END_FUNCTION_BLOCK

// K2/std12k5/TestIm/TestImAlg
	{attribute 'symbol' := 'none'}
FUNCTION_BLOCK TestImAlg EXTENDS BaseAlgoritm
VAR_INPUT
END_VAR
VAR_OUTPUT
END_VAR
VAR
END_VAR

SUPER^();
BlockIm(im:=im.TEN_MB,block:=((BlockOpcControl(block:=FALSE)) OR (im.CMN.onStatus = statusDualInput.STATUS_ERROR) OR (im.CMN.onStatus = statusDualInput.STATUS_NOTDEFINED) OR 
(im.CMN.onStatus = statusDualInput.STATUS_OFF) OR (im.CMN.onStatus = statusDualInput.STATUS_TRANSITIONAL) ));
IF	(im.CMN.onStatus = statusDualInput.STATUS_OFF) AND (im.TEN_MB.onStatus = statusDualInput.STATUS_on) THEN
	im.TEN_MB.off();
END_IF
BlockIm(im:=im.nu.nu1,block:=((BlockOpcControl(block:=FALSE)) OR (im.PNS.onStatus = statusDualInput.STATUS_ERROR) OR (im.pns.onStatus = statusDualInput.STATUS_NOTDEFINED) OR 
(im.pns.onStatus = statusDualInput.STATUS_OFF) OR (im.pns.onStatus = statusDualInput.STATUS_TRANSITIONAL) ));
BlockIm(im:=im.nu.nu2,block:=((BlockOpcControl(block:=FALSE)) OR (im.PNS.onStatus = statusDualInput.STATUS_ERROR) OR (im.pns.onStatus = statusDualInput.STATUS_NOTDEFINED) OR 
(im.pns.onStatus = statusDualInput.STATUS_OFF) OR (im.pns.onStatus = statusDualInput.STATUS_TRANSITIONAL) ));
IF	(im.pns.onStatus = statusDualInput.STATUS_OFF) AND ((im.nu.nu1.onStatus = statusDualInput.STATUS_on) OR (im.nu.nu2.onStatus = statusDualInput.STATUS_on)) THEN
	im.nu.off();
END_IF

METHOD PUBLIC reset
VAR_INPUT
END_VAR
SUPER^.reset();
BlockOpcControl(block:=TRUE);
IF	(algmanager.mode <> modegpa.MODE_AO) AND (algmanager.mode <> modegpa.MODE_NO) AND (algmanager.mode <> modegpa.MODE_EO) THEN
	algManager.setMode(nMode:=ModeGpa.MODE_STOP);
END_IF
im.PNS.DisableOpcControl();
im.nu.nu1.DisableOpcControl();
im.nu.nu2.DisableOpcControl();
im.CMN.DisableOpcControl();
im.TEN_MB.DisableOpcControl();
IF	im.PNS.onStatus = statusDualInput.STATUS_ON THEN
	im.PNS.off();
END_IF
IF	im.nu.nu1.onStatus = statusDualInput.STATUS_ON THEN
	im.nu.nu1.off();
END_IF
IF	im.nu.nu2.onStatus = statusDualInput.STATUS_ON THEN
	im.nu.nu2.off();
END_IF
IF	im.cmn.onStatus = statusDualInput.STATUS_ON THEN
	im.cmn.off();
END_IF
IF	im.TEN_MB.onStatus = statusDualInput.STATUS_ON THEN
	im.TEN_MB.off();
END_IF
END_METHOD

METHOD PUBLIC run
VAR_INPUT
END_VAR
SUPER^.run();
BlockOpcControl(block:=FALSE);
algManager.setMode(nMode:=ModeGpa.MODE_TESTIM);

im.mv.DisableOpcControl ();
im.kran1.DisableOpcControl ();
im.kran2.DisableOpcControl ();
im.kran3.DisableOpcControl ();
im.kran3b.DisableOpcControl ();
im.kran4.DisableOpcControl ();
im.kran5.DisableOpcControl ();
END_METHOD

END_FUNCTION_BLOCK

// K1/std12k5/Start_ALG/Start_NO
{attribute 'symbol' := 'none'}
FUNCTION_BLOCK Start_NO EXTENDS StepBySteapAlgoritm
VAR_INPUT
END_VAR
	
VAR_OUTPUT
	{attribute 'symbol' := 'read'}
	Start_Prov_Pusk:		Question(table:=ADR(ObjectTable)):=			(AnswerVariants:=(Answers.ANS_YES OR Answers.ANS_NO));
END_VAR
VAR
	Alg_Start_reset:	ph_algoritm (table:=ADR(phasesTable)):=		(phaseNumber:=0, Im:=algoritms.no, act:=PhaseAlgoritmAction.run, waitCompletion:=FALSE);
END_VAR

SUPER^();
IF	NOT Alg_Start_reset.start THEN
	Start_Prov_Pusk.ask ();
END_IF
IF	(Start_Prov_Pusk.answer=Answers.ANS_YES) THEN
	algoritms.no.CanRun:=TRUE;
	Alg_Start_reset.run ();
	Start_Prov_Pusk.reset ();
	reset ();
ELSIF	(Start_Prov_Pusk.answer=Answers.ANS_NO) THEN
		algoritms.no.CanRun:=FALSE;
		Start_Prov_Pusk.reset ();
		reset ();
END_IF

METHOD PUBLIC reset
VAR_INPUT
END_VAR
SUPER^.reset();
Start_Prov_Pusk.reset ();
END_METHOD

END_FUNCTION_BLOCK

// K2/std12k5/Start_ALG/Start_NO
{attribute 'symbol' := 'none'}
FUNCTION_BLOCK Start_NO EXTENDS StepBySteapAlgoritm
VAR_INPUT
END_VAR
	
VAR_OUTPUT
	{attribute 'symbol' := 'read'}
	Start_Prov_Pusk:		Question(table:=ADR(ObjectTable)):=			(AnswerVariants:=(Answers.ANS_YES OR Answers.ANS_NO));
END_VAR
VAR
	Alg_Start_reset:	ph_algoritm (table:=ADR(phasesTable)):=		(phaseNumber:=0, Im:=algoritms.no, act:=PhaseAlgoritmAction.run, waitCompletion:=FALSE);
END_VAR

SUPER^();
IF	NOT Alg_Start_reset.start THEN
	Start_Prov_Pusk.ask ();
END_IF
IF	(Start_Prov_Pusk.answer=Answers.ANS_YES) THEN
	algoritms.no.CanRun:=TRUE;
	Alg_Start_reset.run ();
	Start_Prov_Pusk.reset ();
	reset ();
ELSIF	(Start_Prov_Pusk.answer=Answers.ANS_NO) THEN
		algoritms.no.CanRun:=FALSE;
		Start_Prov_Pusk.reset ();
		reset ();
END_IF

METHOD PUBLIC reset
VAR_INPUT
END_VAR
SUPER^.reset();
Start_Prov_Pusk.reset ();
END_METHOD

END_FUNCTION_BLOCK

// K1/std12k5/Start_ALG/Start_AO
{attribute 'symbol' := 'none'}
FUNCTION_BLOCK Start_AO EXTENDS StepBySteapAlgoritm
VAR_INPUT
END_VAR
	
VAR_OUTPUT
	{attribute 'symbol' := 'read'}
	Start_Prov_Pusk:		Question(table:=ADR(ObjectTable)):=			(AnswerVariants:=(Answers.ANS_YES OR Answers.ANS_NO));
END_VAR
VAR
	Alg_Start_reset:	ph_algoritm (table:=ADR(phasesTable)):=		(phaseNumber:=0, Im:=algoritms.ao, act:=PhaseAlgoritmAction.run, waitCompletion:=FALSE);
END_VAR

SUPER^();
IF	NOT Alg_Start_reset.start THEN
	Start_Prov_Pusk.ask ();
END_IF
IF	(Start_Prov_Pusk.answer=Answers.ANS_YES) THEN
	algoritms.ao.CanRun:=TRUE;
	Alg_Start_reset.run ();
	Start_Prov_Pusk.reset ();
	reset ();
ELSIF	(Start_Prov_Pusk.answer=Answers.ANS_NO) THEN
		algoritms.ao.CanRun:=FALSE;
		Start_Prov_Pusk.reset ();
		reset ();
END_IF

METHOD PUBLIC reset
VAR_INPUT
END_VAR
SUPER^.reset();
Start_Prov_Pusk.reset ();
END_METHOD

END_FUNCTION_BLOCK

// K2/std12k5/Start_ALG/Start_AO
{attribute 'symbol' := 'none'}
FUNCTION_BLOCK Start_AO EXTENDS StepBySteapAlgoritm
VAR_INPUT
END_VAR
	
VAR_OUTPUT
	{attribute 'symbol' := 'read'}
	Start_Prov_Pusk:		Question(table:=ADR(ObjectTable)):=			(AnswerVariants:=(Answers.ANS_YES OR Answers.ANS_NO));
END_VAR
VAR
	Alg_Start_reset:	ph_algoritm (table:=ADR(phasesTable)):=		(phaseNumber:=0, Im:=algoritms.ao, act:=PhaseAlgoritmAction.run, waitCompletion:=FALSE);
END_VAR

SUPER^();
IF	NOT Alg_Start_reset.start THEN
	Start_Prov_Pusk.ask ();
END_IF
IF	(Start_Prov_Pusk.answer=Answers.ANS_YES) THEN
	algoritms.ao.CanRun:=TRUE;
	Alg_Start_reset.run ();
	Start_Prov_Pusk.reset ();
	reset ();
ELSIF	(Start_Prov_Pusk.answer=Answers.ANS_NO) THEN
		algoritms.ao.CanRun:=FALSE;
		Start_Prov_Pusk.reset ();
		reset ();
END_IF

METHOD PUBLIC reset
VAR_INPUT
END_VAR
SUPER^.reset();
Start_Prov_Pusk.reset ();
END_METHOD

END_FUNCTION_BLOCK

// K1/std12k5/Logic/SIP_PS
{attribute 'symbol' := 'none'}
FUNCTION_BLOCK SIP_PS EXTENDS BaseIM
VAR_INPUT
	Ai:REFERENCE TO AISource;
END_VAR
VAR_OUTPUT
END_VAR
VAR
	
END_VAR

SUPER^();
IF __ISVALIDREF(Ai) THEN
	
	IF 	ai.interval=statusAi.NOTRELIABLE THEN
		statusSet.setBit (bitNum:=0,value:=1);
	ELSE
		statusSet.setBit (bitNum:=0,value:=0);
	END_IF
END_IF

END_FUNCTION_BLOCK

// K2/std12k5/Logic/SIP_PS
{attribute 'symbol' := 'none'}
FUNCTION_BLOCK SIP_PS EXTENDS BaseIM
VAR_INPUT
	Ai:REFERENCE TO AISource;
END_VAR
VAR_OUTPUT
END_VAR
VAR
	
END_VAR

SUPER^();
IF __ISVALIDREF(Ai) THEN
	
	IF 	ai.interval=statusAi.NOTRELIABLE THEN
		statusSet.setBit (bitNum:=0,value:=1);
	ELSE
		statusSet.setBit (bitNum:=0,value:=0);
	END_IF
END_IF

END_FUNCTION_BLOCK

// K1/std12k5/Ystavki/SIp_Yst
	{attribute 'symbol' := 'none'}
FUNCTION_BLOCK SIp_Yst EXTENDS Baseobject
VAR_INPUT
	{attribute 'symbol' := 'readwright'}
	Yst_izm:ARRAY [0..17] OF UINT;
END_VAR
VAR_OUTPUT
	{attribute 'symbol' := 'read'}
	Yst:ARRAY [0..17] OF UINT;
	
END_VAR
VAR
	flag:BOOL;
	flag2:bool;
	i:uINT;
END_VAR

SUPER^();

FOR i:=0 TO 17 DO
	IF 	(Yst_izm [i] <> Yst [i]) AND (Yst_izm [i] >=0) AND (Yst_izm [i] <=17) THEN
		Yst[i] := Yst_izm [i];
		SaveToFile();
	END_IF	
	
	IF	(Yst_izm [i] = 0) AND (Yst [i] = 0) AND NOT flag AND flag2 THEN
		Yst [i] := 10;
		Yst_izm [i] := Yst [i];
		SaveToFile();
	END_IF


	
END_FOR
IF flag2 THEN
	flag:=TRUE;
END_IF
flag2:=TRUE;

METHOD PROTECTED readPersistent
VAR_INPUT
END_VAR
Yst_izm [0]:=STRING_TO_UINT(readValue());
Yst_izm [1]:=STRING_TO_UINT(readValue());
Yst_izm [2]:=STRING_TO_UINT(readValue());
Yst_izm [3]:=STRING_TO_UINT(readValue());
Yst_izm [4]:=STRING_TO_UINT(readValue());
Yst_izm [5]:=STRING_TO_UINT(readValue());
Yst_izm [6]:=STRING_TO_UINT(readValue());
Yst_izm [7]:=STRING_TO_UINT(readValue());
Yst_izm [8]:=STRING_TO_UINT(readValue());
Yst_izm [9]:=STRING_TO_UINT(readValue());
Yst_izm [10]:=STRING_TO_UINT(readValue());
Yst_izm [11]:=STRING_TO_UINT(readValue());
Yst_izm [12]:=STRING_TO_UINT(readValue());
Yst_izm [13]:=STRING_TO_UINT(readValue());
Yst_izm [14]:=STRING_TO_UINT(readValue());
Yst_izm [15]:=STRING_TO_UINT(readValue());
Yst_izm [16]:=STRING_TO_UINT(readValue());
Yst_izm [17]:=STRING_TO_UINT(readValue());
END_METHOD

METHOD PROTECTED writePersistent
VAR_INPUT
END_VAR

writeValue(value:= UINT_TO_STRING(Yst [0]),'Наработка');
writeValue(value:= UINT_TO_STRING(Yst [1]),'Наработка');
writeValue(value:= UINT_TO_STRING(Yst[2]),'Наработка');
writeValue(value:= UINT_TO_STRING(Yst [3]),'Наработка');

writeValue(value:= UINT_TO_STRING(Yst [4]),'Наработка');
writeValue(value:= UINT_TO_STRING(Yst [5]),'Наработка');
writeValue(value:= UINT_TO_STRING(Yst[6]),'Наработка');
writeValue(value:= UINT_TO_STRING(Yst [7]),'Наработка');

writeValue(value:= UINT_TO_STRING(Yst[8]),'Наработка');
writeValue(value:= UINT_TO_STRING(Yst [9]),'Наработка');
writeValue(value:= UINT_TO_STRING(Yst [10]),'Наработка');
writeValue(value:= UINT_TO_STRING(Yst [11]),'Наработка');

writeValue(value:= UINT_TO_STRING(Yst[12]),'Наработка');
writeValue(value:= UINT_TO_STRING(Yst[13]),'Наработка');
writeValue(value:= UINT_TO_STRING(Yst [14]),'Наработка');
writeValue(value:= UINT_TO_STRING(Yst [15]),'Наработка');
writeValue(value:= UINT_TO_STRING(Yst[16]),'Наработка');
writeValue(value:= UINT_TO_STRING(Yst [17]),'Наработка');
END_METHOD

END_FUNCTION_BLOCK

// K2/std12k5/Ystavki/SIp_Yst
	{attribute 'symbol' := 'none'}
FUNCTION_BLOCK SIp_Yst EXTENDS Baseobject
VAR_INPUT
	{attribute 'symbol' := 'readwright'}
	Yst_izm:ARRAY [0..17] OF UINT;
END_VAR
VAR_OUTPUT
	{attribute 'symbol' := 'read'}
	Yst:ARRAY [0..17] OF UINT;
	
END_VAR
VAR
	flag:BOOL;
	flag2:bool;
	i:uINT;
END_VAR

SUPER^();

FOR i:=0 TO 17 DO
	IF 	(Yst_izm [i] <> Yst [i]) AND (Yst_izm [i] >=0) AND (Yst_izm [i] <=17) THEN
		Yst[i] := Yst_izm [i];
		SaveToFile();
	END_IF	
	
	IF	(Yst_izm [i] = 0) AND (Yst [i] = 0) AND NOT flag AND flag2 THEN
		Yst [i] := 10;
		Yst_izm [i] := Yst [i];
		SaveToFile();
	END_IF


	
END_FOR
IF flag2 THEN
	flag:=TRUE;
END_IF
flag2:=TRUE;

METHOD PROTECTED readPersistent
VAR_INPUT
END_VAR
Yst_izm [0]:=STRING_TO_UINT(readValue());
Yst_izm [1]:=STRING_TO_UINT(readValue());
Yst_izm [2]:=STRING_TO_UINT(readValue());
Yst_izm [3]:=STRING_TO_UINT(readValue());
Yst_izm [4]:=STRING_TO_UINT(readValue());
Yst_izm [5]:=STRING_TO_UINT(readValue());
Yst_izm [6]:=STRING_TO_UINT(readValue());
Yst_izm [7]:=STRING_TO_UINT(readValue());
Yst_izm [8]:=STRING_TO_UINT(readValue());
Yst_izm [9]:=STRING_TO_UINT(readValue());
Yst_izm [10]:=STRING_TO_UINT(readValue());
Yst_izm [11]:=STRING_TO_UINT(readValue());
Yst_izm [12]:=STRING_TO_UINT(readValue());
Yst_izm [13]:=STRING_TO_UINT(readValue());
Yst_izm [14]:=STRING_TO_UINT(readValue());
Yst_izm [15]:=STRING_TO_UINT(readValue());
Yst_izm [16]:=STRING_TO_UINT(readValue());
Yst_izm [17]:=STRING_TO_UINT(readValue());
END_METHOD

METHOD PROTECTED writePersistent
VAR_INPUT
END_VAR

writeValue(value:= UINT_TO_STRING(Yst [0]),'Наработка');
writeValue(value:= UINT_TO_STRING(Yst [1]),'Наработка');
writeValue(value:= UINT_TO_STRING(Yst[2]),'Наработка');
writeValue(value:= UINT_TO_STRING(Yst [3]),'Наработка');

writeValue(value:= UINT_TO_STRING(Yst [4]),'Наработка');
writeValue(value:= UINT_TO_STRING(Yst [5]),'Наработка');
writeValue(value:= UINT_TO_STRING(Yst[6]),'Наработка');
writeValue(value:= UINT_TO_STRING(Yst [7]),'Наработка');

writeValue(value:= UINT_TO_STRING(Yst[8]),'Наработка');
writeValue(value:= UINT_TO_STRING(Yst [9]),'Наработка');
writeValue(value:= UINT_TO_STRING(Yst [10]),'Наработка');
writeValue(value:= UINT_TO_STRING(Yst [11]),'Наработка');

writeValue(value:= UINT_TO_STRING(Yst[12]),'Наработка');
writeValue(value:= UINT_TO_STRING(Yst[13]),'Наработка');
writeValue(value:= UINT_TO_STRING(Yst [14]),'Наработка');
writeValue(value:= UINT_TO_STRING(Yst [15]),'Наработка');
writeValue(value:= UINT_TO_STRING(Yst[16]),'Наработка');
writeValue(value:= UINT_TO_STRING(Yst [17]),'Наработка');
END_METHOD

END_FUNCTION_BLOCK

// K1/std12k5/Narabotka/CMN_
	{attribute 'symbol' := 'none'}
FUNCTION_BLOCK CMN_ EXTENDS nasos
VAR_INPUT
END_VAR
VAR_OUTPUT
		{attribute 'symbol' := 'read'}
	narabotka:UDINT;
		narabotka_:ExtNarabotka (table:=ADR (objectTable)):=(saveInterval:=T#1H);
END_VAR
VAR
	(*timer:RTC;	
	saveTimer:TON:=(PT:=T#600S);
	Narabotka_hour:R_TRIG;
	AvomStartted:R_TRIG;
	narabotka_Izm:UDINT;*)
END_VAR

SUPER^();
narabotka_.started:=onstatus=statusDualInput.STATUS_ON;
narabotka:=(narabotka_.narabotka/3600);
(*
AvomStartted(CLK:=im.CMN.onStatus=statusDualInput.status_on);

	timer.PDT:=UDINT_TO_DT(narabotka_izm);

IF im.CMN.onStatus=statusDualInput.status_on THEN
	narabotka_izm:=DT_TO_UDINT( timer.CDT);
	timer.EN:=TRUE;
ELSE
	timer.EN:=FALSE;
END_IF
narabotka_hour (clk:=(narabotka_izm >=3600));
IF	narabotka_hour.Q THEN
	narabotka:=narabotka+1;
	timer.EN:=FALSE;
	narabotka_izm:=0;
END_IF
timer();

saveTimer(IN:=true);
IF saveTimer.Q THEN
	SaveToFile();
	saveTimer(IN:=FALSE);
END_IF*)

METHOD PROTECTED readPersistent
VAR_INPUT
END_VAR

narabotka:=STRING_TO_UDINT(readValue());
narabotka_izm:=STRING_TO_UDINT(readValue());
END_METHOD

METHOD PROTECTED writePersistent
VAR_INPUT
END_VAR

writeValue(value:= UDINT_TO_STRING(narabotka),'Наработка');
writeValue(value:= UDINT_TO_STRING(narabotka_izm),'Наработка_izm');
END_METHOD

END_FUNCTION_BLOCK

// K2/std12k5/Natabotka/CMN_
	{attribute 'symbol' := 'none'}
FUNCTION_BLOCK CMN_ EXTENDS nasos
VAR_INPUT
END_VAR
VAR_OUTPUT
		{attribute 'symbol' := 'read'}
	narabotka:UDINT;
		narabotka_:ExtNarabotka (table:=ADR (objectTable)):=(saveInterval:=T#1H);
END_VAR
VAR
(*	timer:RTC;	
	saveTimer:TON:=(PT:=T#600S);
	Narabotka_hour:R_TRIG;
	AvomStartted:R_TRIG;
	narabotka_Izm:UDINT;*)
END_VAR

SUPER^();
narabotka_.started:=onstatus=statusDualInput.STATUS_ON;
narabotka:=(narabotka_.narabotka/3600);
(*

AvomStartted(CLK:=im.CMN.onStatus=statusDualInput.status_on);

	timer.PDT:=UDINT_TO_DT(narabotka_izm);

IF im.CMN.onStatus=statusDualInput.status_on THEN
	narabotka_izm:=DT_TO_UDINT( timer.CDT);
	timer.EN:=TRUE;
ELSE
	timer.EN:=FALSE;
END_IF
narabotka_hour (clk:=(narabotka_izm >=3600));
IF	narabotka_hour.Q THEN
	narabotka:=narabotka+1;
	timer.EN:=FALSE;
	narabotka_izm:=0;
END_IF
timer();

saveTimer(IN:=true);
IF saveTimer.Q THEN
	SaveToFile();
	saveTimer(IN:=FALSE);
END_IF*)

METHOD PROTECTED readPersistent
VAR_INPUT
END_VAR

narabotka:=STRING_TO_UDINT(readValue());
narabotka_izm:=STRING_TO_UDINT(readValue());
END_METHOD

METHOD PROTECTED writePersistent
VAR_INPUT
END_VAR

writeValue(value:= UDINT_TO_STRING(narabotka),'Наработка');
writeValue(value:= UDINT_TO_STRING(narabotka_izm),'Наработка_izm');
END_METHOD

END_FUNCTION_BLOCK

// K1/std12k5/Narabotka/Kalorifer_AVOM_
	{attribute 'symbol' := 'none'}
FUNCTION_BLOCK Kalorifer_AVOM_ EXTENDS nasos
VAR_INPUT
END_VAR
VAR_OUTPUT
		{attribute 'symbol' := 'read'}
	narabotka:UDINT;
	narabotka_:ExtNarabotka (table:=ADR (objectTable)):=(saveInterval:=T#1H);
END_VAR
VAR
	(*	timer:RTC;	
	saveTimer:TON:=(PT:=T#600S);
	Narabotka_hour:R_TRIG;
	AvomStartted:R_TRIG;
	narabotka_Izm:UDINT;*)
END_VAR

SUPER^();
narabotka_.started:=onstatus=statusDualInput.STATUS_ON;
narabotka:=(narabotka_.narabotka/3600);
(*
AvomStartted(CLK:=im.KaloriferAVOM.onStatus=statusDualInput.status_on);

	timer.PDT:=UDINT_TO_DT(narabotka_izm);

IF im.KaloriferAVOM.onStatus=statusDualInput.status_on THEN
	narabotka_izm:=DT_TO_UDINT( timer.CDT);
	timer.EN:=TRUE;
ELSE
	timer.EN:=FALSE;
END_IF
narabotka_hour (clk:=(narabotka_izm >=3600));
IF	narabotka_hour.Q THEN
	narabotka:=narabotka+1;
	timer.EN:=FALSE;
	narabotka_izm:=0;
END_IF
timer();

saveTimer(IN:=true);
IF saveTimer.Q THEN
	SaveToFile();
	saveTimer(IN:=FALSE);
END_IF*)

METHOD PROTECTED readPersistent
VAR_INPUT
END_VAR

narabotka:=STRING_TO_UDINT(readValue());
narabotka_izm:=STRING_TO_UDINT(readValue());
END_METHOD

METHOD PROTECTED writePersistent
VAR_INPUT
END_VAR

writeValue(value:= UDINT_TO_STRING(narabotka),'Наработка');
writeValue(value:= UDINT_TO_STRING(narabotka_izm),'Наработка_izm');
END_METHOD

END_FUNCTION_BLOCK

// K2/std12k5/Natabotka/Kalorifer_AVOM_
	{attribute 'symbol' := 'none'}
FUNCTION_BLOCK Kalorifer_AVOM_ EXTENDS nasos
VAR_INPUT
END_VAR
VAR_OUTPUT
		{attribute 'symbol' := 'read'}
	narabotka:UDINT;
	narabotka_:ExtNarabotka (table:=ADR (objectTable)):=(saveInterval:=T#1H);
END_VAR
VAR
	(*	timer:RTC;	
	saveTimer:TON:=(PT:=T#600S);
	Narabotka_hour:R_TRIG;
	AvomStartted:R_TRIG;
	narabotka_Izm:UDINT;*)
END_VAR

SUPER^();
narabotka_.started:=onstatus=statusDualInput.STATUS_ON;
narabotka:=(narabotka_.narabotka/3600);
(*
AvomStartted(CLK:=im.KaloriferAVOM.onStatus=statusDualInput.status_on);

	timer.PDT:=UDINT_TO_DT(narabotka_izm);

IF im.KaloriferAVOM.onStatus=statusDualInput.status_on THEN
	narabotka_izm:=DT_TO_UDINT( timer.CDT);
	timer.EN:=TRUE;
ELSE
	timer.EN:=FALSE;
END_IF
narabotka_hour (clk:=(narabotka_izm >=3600));
IF	narabotka_hour.Q THEN
	narabotka:=narabotka+1;
	timer.EN:=FALSE;
	narabotka_izm:=0;
END_IF
timer();

saveTimer(IN:=true);
IF saveTimer.Q THEN
	SaveToFile();
	saveTimer(IN:=FALSE);
END_IF*)

METHOD PROTECTED readPersistent
VAR_INPUT
END_VAR

narabotka:=STRING_TO_UDINT(readValue());
narabotka_izm:=STRING_TO_UDINT(readValue());
END_METHOD

METHOD PROTECTED writePersistent
VAR_INPUT
END_VAR

writeValue(value:= UDINT_TO_STRING(narabotka),'Наработка');
writeValue(value:= UDINT_TO_STRING(narabotka_izm),'Наработка_izm');
END_METHOD

END_FUNCTION_BLOCK

// K1/std12k5/Narabotka/TEN_Kollectora_
	{attribute 'symbol' := 'none'}
FUNCTION_BLOCK TEN_Kollectora_ EXTENDS nasos
VAR_INPUT
END_VAR
VAR_OUTPUT
		{attribute 'symbol' := 'read'}
	narabotka:UDINT;
	narabotka_:ExtNarabotka (table:=ADR (objectTable)):=(saveInterval:=T#1H);
END_VAR
VAR
(*	timer:RTC;	
	saveTimer:TON:=(PT:=T#600S);
	Narabotka_hour:R_TRIG;
	AvomStartted:R_TRIG;
	narabotka_Izm:UDINT;*)
END_VAR

SUPER^();
narabotka_.started:=onStatus=statusDualInput.STATUS_ON;
narabotka:=(narabotka_.narabotka/3600);
(*
AvomStartted(CLK:=im.TEN_Kollectira.onStatus=statusDualInput.status_on);

	timer.PDT:=UDINT_TO_DT(narabotka_izm);

IF im.TEN_Kollectira.onStatus=statusDualInput.status_on THEN
	narabotka_izm:=DT_TO_UDINT( timer.CDT);
	timer.EN:=TRUE;
ELSE
	timer.EN:=FALSE;
END_IF
narabotka_hour (clk:=(narabotka_izm >=3600));
IF	narabotka_hour.Q THEN
	narabotka:=narabotka+1;
	timer.EN:=FALSE;
	narabotka_izm:=0;
END_IF
timer();

saveTimer(IN:=true);
IF saveTimer.Q THEN
	SaveToFile();
	saveTimer(IN:=FALSE);
END_IF*)

METHOD PROTECTED readPersistent
VAR_INPUT
END_VAR

narabotka:=STRING_TO_UDINT(readValue());
narabotka_izm:=STRING_TO_UDINT(readValue());
END_METHOD

METHOD PROTECTED writePersistent
VAR_INPUT
END_VAR

writeValue(value:= UDINT_TO_STRING(narabotka),'Наработка');
writeValue(value:= UDINT_TO_STRING(narabotka_izm),'Наработка_izm');
END_METHOD

END_FUNCTION_BLOCK

// K2/std12k5/Natabotka/TEN_Kollectora_
	{attribute 'symbol' := 'none'}
FUNCTION_BLOCK TEN_Kollectora_ EXTENDS nasos
VAR_INPUT
END_VAR
VAR_OUTPUT
		{attribute 'symbol' := 'read'}
	narabotka:UDINT;
	narabotka_:ExtNarabotka (table:=ADR (objectTable)):=(saveInterval:=T#1H);
END_VAR
VAR
	(*timer:RTC;	
	saveTimer:TON:=(PT:=T#600S);
	Narabotka_hour:R_TRIG;
	AvomStartted:R_TRIG;
	narabotka_Izm:UDINT;*)
END_VAR

SUPER^();
narabotka_.started:=onStatus=statusDualInput.STATUS_ON;
narabotka:=(narabotka_.narabotka/3600);
(*
AvomStartted(CLK:=im.TEN_Kollectira.onStatus=statusDualInput.status_on);

	timer.PDT:=UDINT_TO_DT(narabotka_izm);

IF im.TEN_Kollectira.onStatus=statusDualInput.status_on THEN
	narabotka_izm:=DT_TO_UDINT( timer.CDT);
	timer.EN:=TRUE;
ELSE
	timer.EN:=FALSE;
END_IF
narabotka_hour (clk:=(narabotka_izm >=3600));
IF	narabotka_hour.Q THEN
	narabotka:=narabotka+1;
	timer.EN:=FALSE;
	narabotka_izm:=0;
END_IF
timer();

saveTimer(IN:=true);
IF saveTimer.Q THEN
	SaveToFile();
	saveTimer(IN:=FALSE);
END_IF*)

METHOD PROTECTED readPersistent
VAR_INPUT
END_VAR

narabotka:=STRING_TO_UDINT(readValue());
narabotka_izm:=STRING_TO_UDINT(readValue());
END_METHOD

METHOD PROTECTED writePersistent
VAR_INPUT
END_VAR

writeValue(value:= UDINT_TO_STRING(narabotka),'Наработка');
writeValue(value:= UDINT_TO_STRING(narabotka_izm),'Наработка_izm');
END_METHOD

END_FUNCTION_BLOCK

// K1/std12k5/Narabotka/TEN_MB_
	{attribute 'symbol' := 'none'}
FUNCTION_BLOCK TEN_MB_ EXTENDS nasos
VAR_INPUT
END_VAR
VAR_OUTPUT
		{attribute 'symbol' := 'read'}
	narabotka:UDINT;
	narabotka_:ExtNarabotka (table:=ADR (objectTable)):=(saveInterval:=T#1H);
END_VAR
VAR
	(*timer:RTC;	
	saveTimer:TON:=(PT:=T#600S);
	Narabotka_hour:R_TRIG;
	AvomStartted:R_TRIG;
	narabotka_Izm:UDINT;*)
END_VAR

SUPER^();
narabotka_.started:=onStatus=statusDualInput.STATUS_ON;
narabotka:=(narabotka_.narabotka/3600);
(*
AvomStartted(CLK:=im.TEN_MB.onStatus=statusDualInput.status_on);

	timer.PDT:=UDINT_TO_DT(narabotka_izm);

IF im.TEN_MB.onStatus=statusDualInput.status_on THEN
	narabotka_izm:=DT_TO_UDINT( timer.CDT);
	timer.EN:=TRUE;
ELSE
	timer.EN:=FALSE;
END_IF
narabotka_hour (clk:=(narabotka_izm >=3600));
IF	narabotka_hour.Q THEN
	narabotka:=narabotka+1;
	timer.EN:=FALSE;
	narabotka_izm:=0;
END_IF
timer();

saveTimer(IN:=true);
IF saveTimer.Q THEN
	SaveToFile();
	saveTimer(IN:=FALSE);
END_IF*)

METHOD PROTECTED readPersistent
VAR_INPUT
END_VAR

narabotka:=STRING_TO_UDINT(readValue());
narabotka_izm:=STRING_TO_UDINT(readValue());
END_METHOD

METHOD PROTECTED writePersistent
VAR_INPUT
END_VAR

writeValue(value:= UDINT_TO_STRING(narabotka),'Наработка');
writeValue(value:= UDINT_TO_STRING(narabotka_izm),'Наработка_izm');
END_METHOD

END_FUNCTION_BLOCK

// K2/std12k5/Natabotka/TEN_MB_
	{attribute 'symbol' := 'none'}
FUNCTION_BLOCK TEN_MB_ EXTENDS nasos
VAR_INPUT
END_VAR
VAR_OUTPUT
		{attribute 'symbol' := 'read'}
	narabotka:UDINT;
	narabotka_:ExtNarabotka (table:=ADR (objectTable)):=(saveInterval:=T#1H);
END_VAR
VAR
	(*timer:RTC;	
	saveTimer:TON:=(PT:=T#600S);
	Narabotka_hour:R_TRIG;
	AvomStartted:R_TRIG;
	narabotka_Izm:UDINT;*)
END_VAR

SUPER^();
narabotka_.started:=onStatus=statusDualInput.STATUS_ON;
narabotka:=(narabotka_.narabotka/3600);
(*
AvomStartted(CLK:=im.TEN_MB.onStatus=statusDualInput.status_on);

	timer.PDT:=UDINT_TO_DT(narabotka_izm);

IF im.TEN_MB.onStatus=statusDualInput.status_on THEN
	narabotka_izm:=DT_TO_UDINT( timer.CDT);
	timer.EN:=TRUE;
ELSE
	timer.EN:=FALSE;
END_IF
narabotka_hour (clk:=(narabotka_izm >=3600));
IF	narabotka_hour.Q THEN
	narabotka:=narabotka+1;
	timer.EN:=FALSE;
	narabotka_izm:=0;
END_IF
timer();

saveTimer(IN:=true);
IF saveTimer.Q THEN
	SaveToFile();
	saveTimer(IN:=FALSE);
END_IF*)

METHOD PROTECTED readPersistent
VAR_INPUT
END_VAR

narabotka:=STRING_TO_UDINT(readValue());
narabotka_izm:=STRING_TO_UDINT(readValue());
END_METHOD

METHOD PROTECTED writePersistent
VAR_INPUT
END_VAR

writeValue(value:= UDINT_TO_STRING(narabotka),'Наработка');
writeValue(value:= UDINT_TO_STRING(narabotka_izm),'Наработка_izm');
END_METHOD

END_FUNCTION_BLOCK

// lowLevel_ecl/im/BaseIms/singleOutput
{attribute 'symbol' := 'none'}
FUNCTION_BLOCK singleOutput EXTENDS BaseIm
VAR_INPUT
	signal:REFERENCE TO BOOL;
	wait_time:TIME:=T#2S;
END_VAR
VAR_OUTPUT
	Q:BOOL;
END_VAR
VAR
	pulseTimer:Ton;
END_VAR
VAR CONSTANT
	cmd_on:WORD:=1;
	cmd_off:WORD:=2;
	cmd_pulse:WORD:=3;
END_VAR

SUPER^();

pulseTimer(PT:=wait_time);
IF pulseTimer.Q THEN
	pulseTimer.IN:=FALSE;
	signal:=FALSE;
END_IF

Q:=signal;
statusSet.setBit(0,Q);

METHOD on
VAR_INPUT
END_VAR
setCmd(nCmd:=cmd_on);
signal:=TRUE;
resetCommand();
END_METHOD

METHOD PROTECTED processCmd;
VAR_INPUT
	cmd:UINT;
	sender:UINT;
	parametr:UINT;
END_VAR
SUPER^.processCmd(cmd,sender,parametr);
CASE cmd OF
	cmd_on:on();
	cmd_off:off();
	cmd_pulse:impulse();
END_CASE
END_METHOD

METHOD impulse
VAR_INPUT
	
END_VAR
setCmd(nCmd:=cmd_on);
signal:=TRUE;
pulseTimer.IN:=TRUE;
END_METHOD

METHOD off
VAR_INPUT
END_VAR
setCmd(nCmd:=cmd_off);
signal:=FALSE;
pulseTimer.IN:=FALSE;
resetCommand();
END_METHOD

END_FUNCTION_BLOCK

// K2/std12k5/Ystavki/AutoPNS_YP
	{attribute 'symbol' := 'none'}
FUNCTION_BLOCK AutoPNS_YP EXTENDS Baseobject
VAR_INPUT
	{attribute 'symbol' := 'readwright'}
	Yst_izm:UDINT;
END_VAR
VAR_OUTPUT
	
	{attribute 'symbol' := 'read'}
	Yst:UDINT;
	
END_VAR
VAR
	Yst_Izm_trig:R_TRIG;
	Yst_First_izm:R_TRIG;
	flag:bool;
END_VAR

SUPER^();

Yst_Izm_trig (clk:=((Yst_izm <> Yst) 	AND (Yst_izm >0) AND (Yst_izm < 1000) AND (Yst_izm < Ystavki.YstPNS_YT.Yst)));
IF 	Yst_Izm_trig.Q THEN
	Yst := Yst_izm;
	SaveToFile();
END_IF
Yst_First_izm (clk:= ((Yst_izm = 0) AND (Yst = 0) AND flag ));
IF	Yst_First_izm.Q  THEN
	Yst := 300;
	Yst_izm := Yst;
	SaveToFile();
END_IF;
flag:=TRUE;

METHOD PROTECTED readPersistent
VAR_INPUT
END_VAR
Yst_izm:=STRING_TO_UDINT(readValue());
END_METHOD

METHOD PROTECTED writePersistent
VAR_INPUT
END_VAR
writeValue(value:= UDINT_TO_STRING(Yst),'Наработка');
END_METHOD

END_FUNCTION_BLOCK

// K1/std12k5/Ystavki/AutoPNS_YP
	{attribute 'symbol' := 'none'}
FUNCTION_BLOCK AutoPNS_YP EXTENDS Baseobject
VAR_INPUT
	{attribute 'symbol' := 'readwright'}
	Yst_izm:UDINT;
END_VAR
VAR_OUTPUT
	
	{attribute 'symbol' := 'read'}
	Yst:UDINT;
	
END_VAR
VAR
	Yst_Izm_trig:R_TRIG;
	Yst_First_izm:R_TRIG;
	flag:bool;
END_VAR

SUPER^();

Yst_Izm_trig (clk:=((Yst_izm <> Yst) 	AND (Yst_izm >0) AND (Yst_izm < 1000) AND (Yst_izm < Ystavki.YstPNS_YT.Yst)));
IF 	Yst_Izm_trig.Q THEN
	Yst := Yst_izm;
	SaveToFile();
END_IF
Yst_First_izm (clk:= ((Yst_izm = 0) AND (Yst = 0) AND flag ));
IF	Yst_First_izm.Q  THEN
	Yst := 300;
	Yst_izm := Yst;
	SaveToFile();
END_IF;
flag:=TRUE;

METHOD PROTECTED readPersistent
VAR_INPUT
END_VAR
Yst_izm:=STRING_TO_UDINT(readValue());
END_METHOD

METHOD PROTECTED writePersistent
VAR_INPUT
END_VAR
writeValue(value:= UDINT_TO_STRING(Yst),'Наработка');
END_METHOD

END_FUNCTION_BLOCK

// K2/std12k5/TestIm/Imit_OPC
{attribute 'symbol' := 'none'}
FUNCTION_BLOCK Imit_OPC EXTENDS BaseAlgoritm
VAR_INPUT
END_VAR
	
VAR_OUTPUT
	
	OPC_block_izm:uINT;
END_VAR
VAR
	
END_VAR

SUPER^();
IF (OPC_block_izm <> ystavki.block_OPC_cmd.Value) AND kontroller.imit THEN
IF 	ystavki.block_OPC_cmd.Value = 1 THEN
	im.kran1.EnableOpcControl ();
	im.kran2.EnableOpcControl ();
	im.kran3.EnableOpcControl ();
	im.kran3b.EnableOpcControl ();
	im.kran4.EnableOpcControl ();
	im.kran5.EnableOpcControl ();
	im.kran6.EnableOpcControl ();
	im.PNS.EnableOpcControl ();
	im.nu.nu1.EnableOpcControl ();
	im.nu.nu2.EnableOpcControl ();
	im.CMN.EnableOpcControl ();
	im.TEN_Kollectira.EnableOpcControl ();
	im.TEN_MB.EnableOpcControl ();
	im.KaloriferAVOM.EnableOpcControl ();
	im.v1_Avom.EnableOpcControl ();
	im.v2_Avom.EnableOpcControl ();
	im.v3_Avom.EnableOpcControl ();
	im.v4_Avom.EnableOpcControl ();
	im.mv.EnableOpcControl ();
ELSE
	im.kran1.DisableOpcControl ();
	im.kran2.DisableOpcControl ();
	im.kran3.DisableOpcControl ();
	im.kran3b.DisableOpcControl ();
	im.kran4.DisableOpcControl ();
	im.kran5.DisableOpcControl ();
	im.kran6.DisableOpcControl ();
	im.PNS.DisableOpcControl ();
	im.nu.nu1.DisableOpcControl ();
	im.nu.nu2.DisableOpcControl ();
	im.CMN.DisableOpcControl ();
	im.TEN_Kollectira.DisableOpcControl ();
	im.TEN_MB.DisableOpcControl ();
	im.KaloriferAVOM.DisableOpcControl ();
	im.v1_Avom.DisableOpcControl ();
	im.v2_Avom.DisableOpcControl ();
	im.v3_Avom.DisableOpcControl ();
	im.v4_Avom.DisableOpcControl ();
	im.mv.DisableOpcControl ();
END_IF
END_IF

OPC_block_izm :=ystavki.block_OPC_cmd.Value;

END_FUNCTION_BLOCK

// K1/std12k5/TestIm/Imit_OPC
{attribute 'symbol' := 'none'}
FUNCTION_BLOCK Imit_OPC EXTENDS BaseAlgoritm
VAR_INPUT
END_VAR
	
VAR_OUTPUT
	
	OPC_block_izm:uINT;
END_VAR
VAR
	
END_VAR

SUPER^();
IF (OPC_block_izm <> ystavki.block_OPC_cmd.Value) AND kontroller.imit THEN
IF 	ystavki.block_OPC_cmd.Value = 1 THEN
	im.kran1.EnableOpcControl ();
	im.kran2.EnableOpcControl ();
	im.kran3.EnableOpcControl ();
	im.kran3b.EnableOpcControl ();
	im.kran4.EnableOpcControl ();
	im.kran5.EnableOpcControl ();
	im.kran6.EnableOpcControl ();
	im.PNS.EnableOpcControl ();
	im.nu.nu1.EnableOpcControl ();
	im.nu.nu2.EnableOpcControl ();
	im.CMN.EnableOpcControl ();
	im.TEN_Kollectira.EnableOpcControl ();
	im.TEN_MB.EnableOpcControl ();
	im.KaloriferAVOM.EnableOpcControl ();
	im.v1_Avom.EnableOpcControl ();
	im.v2_Avom.EnableOpcControl ();
	im.v3_Avom.EnableOpcControl ();
	im.v4_Avom.EnableOpcControl ();
	im.mv.EnableOpcControl ();
ELSE
	im.kran1.DisableOpcControl ();
	im.kran2.DisableOpcControl ();
	im.kran3.DisableOpcControl ();
	im.kran3b.DisableOpcControl ();
	im.kran4.DisableOpcControl ();
	im.kran5.DisableOpcControl ();
	im.kran6.DisableOpcControl ();
	im.PNS.DisableOpcControl ();
	im.nu.nu1.DisableOpcControl ();
	im.nu.nu2.DisableOpcControl ();
	im.CMN.DisableOpcControl ();
	im.TEN_Kollectira.DisableOpcControl ();
	im.TEN_MB.DisableOpcControl ();
	im.KaloriferAVOM.DisableOpcControl ();
	im.v1_Avom.DisableOpcControl ();
	im.v2_Avom.DisableOpcControl ();
	im.v3_Avom.DisableOpcControl ();
	im.v4_Avom.DisableOpcControl ();
	im.mv.DisableOpcControl ();
END_IF
END_IF

OPC_block_izm :=ystavki.block_OPC_cmd.Value;

END_FUNCTION_BLOCK

// LowLevel_Algoritms/im/Reability
{attribute 'symbol' := 'none'}
FUNCTION_BLOCK Reability EXTENDS BaseIm
VAR_INPUT
	di1:REFERENCE TO reliablebit;
	
END_VAR 
VAR_OUTPUT
END_VAR
VAR
	when:bool;
END_VAR

SUPER^();
IF __ISVALIDREF(di1)  THEN
	IF when THEN
		IF	(di1.reliability = 1) THEN
			statusSet.setBit (bitNum:=0,value:=1);
	
		ELSE
			statusSet.setBit (bitNum:=0,value:=0);
		END_IF
	ELSE
		IF	(di1.reliability = 0) THEN
			statusSet.setBit (bitNum:=0,value:=1);
		ELSE
			statusSet.setBit (bitNum:=0,value:=0);
		END_IF
	end_if;
END_IF

END_FUNCTION_BLOCK

// lowLevel_ecl/algoritms/phases/ph_Analog
	{attribute 'symbol' := 'none'}
	{attribute 'obsolete' := 'Have unsafe interface. Use WaitAnalogValue. '} 
FUNCTION_BLOCK ph_Analog EXTENDS BaseAlgoritmPhase
VAR_INPUT
	ai:REFERENCE TO AISource;
	more_param:REFERENCE TO AnalogParametr;
	less_param:REFERENCE TO AnalogParametr;
	more:REAL:=RNaN();
	less:REAL:=RNaN();	
END_VAR
VAR_OUTPUT
END_VAR
VAR
END_VAR

SUPER^();

METHOD PROTECTED getError : bool
VAR_INPUT
END_VAR
getError:=ai.interval<statusAi.normal;
END_METHOD

METHOD protected GetIm : POINTER TO BaseIm
VAR_INPUT
END_VAR
GetIm:=adr(ai);
END_METHOD

METHOD PROTECTED getTop : bool
VAR_INPUT
END_VAR
IF (ai.interval<statusAi.normal) THEN
	getTop:=FALSE;
	RETURN;
END_IF

IF __ISVALIDREF(more_param) OR __ISVALIDREF(less_param) THEN
	getTop:=TRUE;
	IF  __ISVALIDREF(more_param) THEN
		getTop:=getTop AND (ai.value>more_param.Value);	
	END_IF
	
	IF __ISVALIDREF(less_param) THEN
		getTop:=getTop AND (ai.value<less_param.Value);	
	END_IF	
ELSIF (NOT FPU.IsRealNaN(more)) OR (NOT FPU.IsRealNaN(less)) THEN
	getTop:=TRUE;
	IF  NOT FPU.IsRealNaN(more) THEN
		getTop:=getTop AND (ai.value>more);	
	END_IF
	
	IF NOT FPU.IsRealNaN(less) THEN
		getTop:=getTop AND (ai.value<less);	
	END_IF	
ELSE
	getTop:=TRUE;	
END_IF
END_METHOD

METHOD PROTECTED onRun
VAR_INPUT
END_VAR
SUPER^.onRun();
END_METHOD

END_FUNCTION_BLOCK

// lowLevel_ecl/algoritms/phases/ph_SingleOutput
	{attribute 'symbol' := 'none'}
FUNCTION_BLOCK ph_SingleOutput EXTENDS BaseAlgoritmPhase
VAR_INPUT
	Im:REFERENCE TO singleOutput;
	WhatCanIdo:BOOL;
END_VAR
VAR_OUTPUT
END_VAR
VAR
END_VAR

SUPER^();

METHOD PROTECTED getError : bool
VAR_INPUT
END_VAR
END_METHOD

METHOD protected GetIm : POINTER TO BaseIm
VAR_INPUT
END_VAR
GetIm:=adr(Im);
END_METHOD

METHOD PROTECTED getTop : bool
VAR_INPUT
END_VAR
getTop:=Im.Q=WhatCanIdo;
END_METHOD

METHOD PROTECTED onRun
VAR_INPUT
END_VAR
IF (WhatCanIdo) THEN
	Im.on();
ELSE
	Im.off();
END_IF
END_METHOD

END_FUNCTION_BLOCK

// lowLevel_ecl/algoritms/phases/ph_WaitAnalogValue
	{attribute 'symbol' := 'none'}
FUNCTION_BLOCK ph_WaitAnalogValue EXTENDS BaseAlgoritmPhase
VAR_INPUT
	ai:REFERENCE TO AISource;
	more:IAnalogValue;
	less:IAnalogValue;	
END_VAR
VAR_OUTPUT
END_VAR
VAR
END_VAR

SUPER^();

METHOD PROTECTED getError : bool
VAR_INPUT
END_VAR
getError:=ai.interval<statusAi.normal;
END_METHOD

METHOD protected GetIm : POINTER TO BaseIm
VAR_INPUT
END_VAR
GetIm:=adr(ai);
END_METHOD

METHOD PROTECTED getTop : bool
VAR_INPUT
END_VAR
IF (ai.interval<statusAi.normal) THEN
	getTop:=FALSE;
	RETURN;
END_IF

IF (more<>0) OR (less<>0) THEN
	getTop:=TRUE;
	IF  more<>0 THEN
		getTop:=getTop AND (ai.value>more.getValue());	
	END_IF
	
	IF less<>0 THEN
		getTop:=getTop AND (ai.value<less.getValue());	
	END_IF	
ELSE
	getTop:=TRUE;	
END_IF
END_METHOD

METHOD PROTECTED onRun
VAR_INPUT
END_VAR
SUPER^.onRun();
END_METHOD

END_FUNCTION_BLOCK

// lowLevel_ecl/algoritms/runAlg
FUNCTION runAlg : BOOL
VAR_INPUT
	alg:REFERENCE TO BaseAlgoritm;
END_VAR
VAR
END_VAR

IF __ISVALIDREF(alg) THEN
	IF NOT alg.isRuning THEN
		alg.run();
	END_IF;
END_IF;

END_FUNCTION

// K1/std12k5/Logic/All_Quation_Off
	{attribute 'symbol' := 'none'}
FUNCTION_BLOCK All_Quation_Off EXTENDS Question
VAR_INPUT
END_VAR
VAR_OUTPUT
	
	
END_VAR
VAR
	
	ton1:ton ;
	ton2:ton ;
	ton3:ton ;
END_VAR

SUPER^();
algoritms.Opres.Zapolnit_kontur.resetAns(in:=TRUE, PT:=T#0S);
algoritms.Opres.PNS_NU_ON_Ask.resetAns(in:=TRUE, PT:=T#0S);
algoritms.Opres.Opressovka_Start.resetAns(in:=TRUE, PT:=T#0S);
algoritms.autoNu_1.NU_OFF_Ask.resetAns(in:=TRUE, PT:=T#0S);
algoritms.autoNu_2.NU_osn_OFF_Ask.resetAns(in:=TRUE, PT:=T#0S);
algoritms.autoNu_2.NU_rez_OFF_Ask.resetAns(in:=TRUE, PT:=T#0S);
algoritms.autoPns.PNS_Off.resetAns(in:=TRUE, PT:=T#0S);
algoritms.ao.sbrosVibeg.resetAns(in:=TRUE, PT:=T#0S);
algoritms.no.sbrosVibeg.resetAns(in:=TRUE, PT:=T#0S);
algoritms.dPmg.NU_OFF_Ask.resetAns(in:=TRUE, PT:=T#0S);
algoritms.Pms.PNS_OFF_Ask.resetAns(in:=TRUE, PT:=T#0S);
algoritms.F4.Kr_12_Move.resetAns(in:=TRUE, PT:=T#0S);
algoritms.AutoPNS_Start.AutoPNS_Ask.resetAns(in:=TRUE, PT:=T#0S);
algoritms.R_AutoAVom.Start_Prov_Pusk.resetAns(in:=TRUE, PT:=T#0S);
algoritms.R_AutoTEN.Start_Prov_Pusk.resetAns(in:=TRUE, PT:=T#0S);
algoritms.R_TestIM.Start_Prov_Pusk.resetAns(in:=TRUE, PT:=T#0S);
algoritms.S_AO.Start_Prov_Pusk.resetAns(in:=TRUE, PT:=T#0S);
algoritms.S_AutoAVOM.Start_Prov_Pusk.resetAns(in:=TRUE, PT:=T#0S);
algoritms.S_AutoTEN.Start_Prov_Pusk.resetAns(in:=TRUE, PT:=T#0S);
algoritms.S_NO.Start_Prov_Pusk.resetAns(in:=TRUE, PT:=T#0S);
algoritms.S_dPmg.Start_Prov_Pusk.resetAns(in:=TRUE, PT:=T#0S);
algoritms.S_I.Start_Prov_Pusk.resetAns(in:=TRUE, PT:=T#0S);
algoritms.S_K.Start_Prov_Pusk.resetAns(in:=TRUE, PT:=T#0S);
algoritms.S_K.F4_Start_Q.resetAns(in:=TRUE, PT:=T#0S);
algoritms.S_Pms.Start_Prov_Pusk.resetAns(in:=TRUE, PT:=T#0S);
algoritms.S_V.Start_Prov_Pusk.resetAns(in:=TRUE, PT:=T#0S);
algoritms.S_AP.Start_Prov_Pusk.resetAns(in:=TRUE, PT:=T#0S);
algoritms.S_PP.Start_Prov_Pusk.resetAns(in:=TRUE, PT:=T#0S);
algoritms.S_PP.F2_Ask.resetAns(in:=TRUE, PT:=T#0S);
algoritms.S_PP.F3_Ask.resetAns(in:=TRUE, PT:=T#0S);
algoritms.S_PP.F4_Ask.resetAns(in:=TRUE, PT:=T#0S);
algoritms.S_Test_IM.Start_Prov_Pusk.resetAns(in:=TRUE, PT:=T#0S);

END_FUNCTION_BLOCK

// K2/std12k5/Logic/All_Quation_Off
	{attribute 'symbol' := 'none'}
FUNCTION_BLOCK All_Quation_Off EXTENDS Question
VAR_INPUT
END_VAR
VAR_OUTPUT
	
	
END_VAR
VAR
	
	ton1:ton ;
	ton2:ton ;
	ton3:ton ;
END_VAR

SUPER^();
algoritms.Opres.Zapolnit_kontur.resetAns(in:=TRUE, PT:=T#0S);
algoritms.Opres.PNS_NU_ON_Ask.resetAns(in:=TRUE, PT:=T#0S);
algoritms.Opres.Opressovka_Start.resetAns(in:=TRUE, PT:=T#0S);
algoritms.autoNu_1.NU_OFF_Ask.resetAns(in:=TRUE, PT:=T#0S);
algoritms.autoNu_2.NU_osn_OFF_Ask.resetAns(in:=TRUE, PT:=T#0S);
algoritms.autoNu_2.NU_rez_OFF_Ask.resetAns(in:=TRUE, PT:=T#0S);
algoritms.autoPns.PNS_Off.resetAns(in:=TRUE, PT:=T#0S);
algoritms.ao.sbrosVibeg.resetAns(in:=TRUE, PT:=T#0S);
algoritms.no.sbrosVibeg.resetAns(in:=TRUE, PT:=T#0S);
algoritms.dPmg.NU_OFF_Ask.resetAns(in:=TRUE, PT:=T#0S);
algoritms.Pms.PNS_OFF_Ask.resetAns(in:=TRUE, PT:=T#0S);
algoritms.F4.Kr_12_Move.resetAns(in:=TRUE, PT:=T#0S);
algoritms.AutoPNS_Start.AutoPNS_Ask.resetAns(in:=TRUE, PT:=T#0S);
algoritms.R_AutoAVom.Start_Prov_Pusk.resetAns(in:=TRUE, PT:=T#0S);
algoritms.R_AutoTEN.Start_Prov_Pusk.resetAns(in:=TRUE, PT:=T#0S);
algoritms.R_TestIM.Start_Prov_Pusk.resetAns(in:=TRUE, PT:=T#0S);
algoritms.S_AO.Start_Prov_Pusk.resetAns(in:=TRUE, PT:=T#0S);
algoritms.S_AutoAVOM.Start_Prov_Pusk.resetAns(in:=TRUE, PT:=T#0S);
algoritms.S_AutoTEN.Start_Prov_Pusk.resetAns(in:=TRUE, PT:=T#0S);
algoritms.S_NO.Start_Prov_Pusk.resetAns(in:=TRUE, PT:=T#0S);
algoritms.S_dPmg.Start_Prov_Pusk.resetAns(in:=TRUE, PT:=T#0S);
algoritms.S_I.Start_Prov_Pusk.resetAns(in:=TRUE, PT:=T#0S);
algoritms.S_K.Start_Prov_Pusk.resetAns(in:=TRUE, PT:=T#0S);
algoritms.S_K.F4_Start_Q.resetAns(in:=TRUE, PT:=T#0S);
algoritms.S_Pms.Start_Prov_Pusk.resetAns(in:=TRUE, PT:=T#0S);
algoritms.S_V.Start_Prov_Pusk.resetAns(in:=TRUE, PT:=T#0S);
algoritms.S_AP.Start_Prov_Pusk.resetAns(in:=TRUE, PT:=T#0S);
algoritms.S_PP.Start_Prov_Pusk.resetAns(in:=TRUE, PT:=T#0S);
algoritms.S_PP.F2_Ask.resetAns(in:=TRUE, PT:=T#0S);
algoritms.S_PP.F3_Ask.resetAns(in:=TRUE, PT:=T#0S);
algoritms.S_PP.F4_Ask.resetAns(in:=TRUE, PT:=T#0S);
algoritms.S_Test_IM.Start_Prov_Pusk.resetAns(in:=TRUE, PT:=T#0S);

END_FUNCTION_BLOCK

// lowLevel_ecl/im/ventvs/Switch
	{attribute 'symbol' := 'none'}
FUNCTION_BLOCK PUBLIC Switch EXTENDS Ventvs
VAR_INPUT

END_VAR
VAR_OUTPUT

END_VAR
VAR
END_VAR

SUPER^();

END_FUNCTION_BLOCK

// lowLevel_ecl/im/ventvs/Zaslonka
	{attribute 'symbol' := 'none'}
FUNCTION_BLOCK Zaslonka EXTENDS Ventvs
VAR_INPUT
END_VAR
VAR_OUTPUT
END_VAR
VAR
END_VAR

SUPER^();

END_FUNCTION_BLOCK

// lowLevel_ecl/im/Zadvigka/Zadvigka
	{attribute 'symbol' := 'none'}
FUNCTION_BLOCK Zadvigka EXTENDS DualStateKran
VAR_INPUT
	inLocal: REFERENCE TO ReliableBit;	
	inDistance: REFERENCE TO ReliableBit;
	inAuto:REFERENCE TO ReliableBit;
	inManual: REFERENCE TO ReliableBit;
	
	inErrorPowerOff: REFERENCE TO ReliableBit;
	inErrorBlock: REFERENCE TO ReliableBit;	

END_VAR
VAR_OUTPUT

END_VAR
VAR
	Local: BOOL;	
	Distance: BOOL;
	Auto:BOOL;
	Manual:BOOL;
	
	ErrorPowerOff: BOOL;
	ErrorBlock: BOOL;	
END_VAR

SUPER^();
Local:=checkArg(inLocal);
Distance:=checkArg(inDistance);
Auto:=checkArg(inAuto);
Manual:=checkArg(inManual);

ErrorPowerOff:=checkArg(inErrorPowerOff);
ErrorBlock:=checkArg(inErrorBlock);

METHOD PROTECTED getSdvig : BOOL
VAR_INPUT
END_VAR
getSdvig:=FALSE;
IF (NOT Local) THEN
	getSdvig:=super^.getSdvig();
END_IF
END_METHOD

METHOD PUBLIC writeImStatus
VAR_INPUT
END_VAR
SUPER^.writeImStatus();
statusSet.setBit(5,Local);
statusSet.setBit(6,Distance);
statusSet.setBit(7,Auto);
statusSet.setBit(8,Manual);

statusSet.setBit(10,ErrorPowerOff);
statusSet.setBit(11,ErrorBlock);
END_METHOD

END_FUNCTION_BLOCK

// lowLevel_ecl/kontroller/modbus/MlpMbKontroller
{attribute 'symbol' := 'none'}
FUNCTION_BLOCK MlpMbKontroller EXTENDS MbKontroller
VAR_INPUT
	mlp:REFERENCE TO Elpk04;
	DinStartAddr:INT;
	DoutStartAddr:INT;
END_VAR
VAR_OUTPUT

END_VAR
VAR

END_VAR

SUPER^();

METHOD PUBLIC getInputFloat : REAL
VAR_INPUT
	addr:WORD;
END_VAR
VAR
	rawValue:FloatAsWords;
END_VAR
CASE AiWordOrder OF
	MbAiWordOrder.AiWordOrder12:
		rawValue.wValue[0]:=getInputValue(addr:=addr);
		rawValue.wValue[1]:=getInputValue(addr:=addr+1);	
	MbAiWordOrder.AiWordOrder21:
		rawValue.wValue[0]:=getInputValue(addr:=addr+1);
		rawValue.wValue[1]:=getInputValue(addr:=addr);
END_CASE

getInputFloat:=rawValue.fValue;
END_METHOD

METHOD PUBLIC getInputValue : WORD
VAR_INPUT
	addr:WORD;
END_VAR
getInputValue:=mlp.DIn_[DinStartAddr+addr].val;
END_METHOD

METHOD PUBLIC setOutputByte
VAR_INPUT
	addr:WORD;
	value:BYTE;
	usedByte:UsedByteMBSource;
END_VAR
VAR
	rawValue:FloatAsWords;
	
END_VAR
rawValue.wValue[0]:=	holding[addr]; // сохраняем 
IF usedByte=UsedByteMBSource.HB THEN 
	rawValue.bValue[1]:=	value;
ELSE
	rawValue.bValue[0]:=	value;
END_IF
mlp.Dout_[DoutStartAddr+addr]:=rawValue.wValue[0]; //кормим слово
END_METHOD

METHOD PUBLIC setOutputFloat
VAR_INPUT
	addr:WORD;
	value:REAL;
END_VAR
VAR
	rawValue:FloatAsWords;
END_VAR
rawValue.fValue:=value;
CASE AiWordOrder OF
	MbAiWordOrder.AiWordOrder12:
		setOutputValue(addr:=addr,value:=rawValue.wValue[0]);
		setOutputValue(addr:=addr+1,value:=rawValue.wValue[1]);	
	MbAiWordOrder.AiWordOrder21:
		setOutputValue(addr:=addr+1,value:=rawValue.wValue[0]);
		setOutputValue(addr:=addr,value:=rawValue.wValue[1]);	
END_CASE
END_METHOD

METHOD PUBLIC setOutputValue
VAR_INPUT
	addr:WORD;
	value:WORD;
END_VAR
mlp.Dout_[DoutStartAddr+addr]:=value;
END_METHOD

END_FUNCTION_BLOCK

// lowLevel_ecl/kontroller/modbus/Sources/DoSourceMb
{attribute 'symbol' := 'none'}
FUNCTION_BLOCK DoSourceMb EXTENDS DOSource
IMPLEMENTS IMbSource;
VAR_INPUT
	
END_VAR
VAR_OUTPUT
END_VAR
VAR
	mbKontr:REFERENCE TO MbKontroller;
	bitNumber:int;
END_VAR

SUPER^();

METHOD setKontroller
VAR_INPUT
	nKontroller	: REFERENCE TO MbKontroller;
END_VAR
mbKontr REF=nKontroller;
END_METHOD

METHOD writeData
VAR_INPUT
	value:WORD;
END_VAR
mbKontr.setOutputValue(addr:=addr,value:=value);
END_METHOD

END_FUNCTION_BLOCK

// lowLevel_ecl/kontroller/modbus/Sources/SpecSources/AiSourceMbByte
{attribute 'symbol' := 'none'}
FUNCTION_BLOCK AiSourceMbByte EXTENDS AiSourceMb
VAR_INPUT
	usedByte:UsedByteMBSource;
END_VAR
VAR_OUTPUT
END_VAR
VAR
END_VAR

SUPER^();

METHOD PROTECTED GetData : Real
VAR_INPUT
END_VAR
VAR_OUTPUT
	o_interval:statusAi;
END_VAR
VAR
	rawValue:FloatAsWords;
	realValue:REAL;
END_VAR
 rawValue.wValue[0]:=mbKontr.getInputValue(addr:=addr);

CASE usedByte OF
	UsedByteMBSource.LB: realValue:=BYTE_TO_REAL(rawValue.bValue[0]);
	UsedByteMBSource.HB: realValue:=BYTE_TO_REAL(rawValue.bValue[1]);
END_CASE

source.input:=realValue;
source.k:=k;
source.b:=b;
source.h:=histeresis;
source.ap:=aperturFilter;
source.dp:=pikFiler;
source.ds:=exponentialFilter;
source.de:=rassoglasovanie;
source();

GetData:=source.value;

IF __ISVALIDREF(reliability) THEN
	IF reliability.reliability AND reliability.value THEN
		o_interval:=statusAi.normal;
	ELSE
		o_interval:=statusAi.NOTDEFINED;
	END_IF
ELSE
	o_interval:=statusAi.normal;	
END_IF
END_METHOD

END_FUNCTION_BLOCK

// lowLevel_ecl/kontroller/modbus/Sources/SpecSources/AiSourceMbWord
{attribute 'symbol' := 'none'}
FUNCTION_BLOCK AiSourceMbWord EXTENDS AiSourceMb
VAR_INPUT
END_VAR
VAR_OUTPUT
END_VAR
VAR
END_VAR

SUPER^();

METHOD PROTECTED GetData : Real
VAR_INPUT
END_VAR
VAR_OUTPUT
	o_interval:statusAi;
END_VAR
VAR
	rawValue:FloatAsWords;
	realValue:REAL;
END_VAR
rawValue.wValue[0]:=mbKontr.getInputValue(addr:=addr);
source.input:=rawValue.wValue[0];
source.k:=k;
source.b:=b;
source.h:=histeresis;
source.ap:=aperturFilter;
source.dp:=pikFiler;
source.ds:=exponentialFilter;
source.de:=rassoglasovanie;
source();

IF rawValue.wValue[0] < 16#7FFD THEN  // ограничение на макс значение
GetData:=source.value;

IF __ISVALIDREF(reliability) THEN
	IF reliability.reliability AND reliability.value THEN
		o_interval:=statusAi.normal;
	ELSE
		o_interval:=statusAi.NOTDEFINED;
	END_IF
ELSE
	o_interval:=statusAi.normal;	
END_IF
ELSE
o_interval:=statusAi.NOTDEFINED;
END_IF
END_METHOD

END_FUNCTION_BLOCK

// lowLevel_ecl/kontroller/modbus/Sources/SpecSources/AoProxiMbByte
{attribute 'symbol' := 'none'}
FUNCTION_BLOCK AoProxiMbByte  EXTENDS AoProxiMb
VAR_INPUT
		usedByte:UsedByteMBSource;
END_VAR
VAR_OUTPUT
END_VAR
VAR
END_VAR

SUPER^();

METHOD PROTECTED writeData
VAR_INPUT
	val:REAL;
END_VAR
VAR

END_VAR
mbKontr.setOutputByte(addr:=addr,value:=REAL_TO_BYTE(k*Value+b)	,usedByte:=usedByte);
END_METHOD

END_FUNCTION_BLOCK

// lowLevel_ecl/kontroller/modbus/Sources/SpecSources/AoProxiMbWord
{attribute 'symbol' := 'none'}
FUNCTION_BLOCK AoProxiMbWord  EXTENDS AoProxiMb
VAR_INPUT
		usedByte:UsedByteMBSource;
END_VAR
VAR_OUTPUT
END_VAR
VAR
END_VAR

SUPER^();

METHOD PROTECTED writeData
VAR_INPUT
	val:REAL;
END_VAR
VAR
	rawValue:FloatAsWords;	
END_VAR
IF __ISVALIDREF(Source) THEN
	rawValue.fValue:=Source.value;
	mbKontr.setOutputValue(addr:=addr+1,value:=Source.interval);
ELSE
	rawValue.fValue:=k*Value+b;	
END_IF
rawValue.wValue[0]:= REAL_TO_WORD(rawValue.fValue);
mbKontr.setOutputValue(addr:=addr,value:=rawValue.wValue[0]);
END_METHOD

END_FUNCTION_BLOCK

// K2/std12k5/Start_ALG/Start_Test_Pr
{attribute 'symbol' := 'none'}
FUNCTION_BLOCK Start_Test_Pr EXTENDS StepBySteapAlgoritm
VAR_INPUT
END_VAR
	
VAR_OUTPUT
	{attribute 'symbol' := 'read'}
	Start_Prov_Pusk:		Question(table:=ADR(ObjectTable)):=			(AnswerVariants:=(Answers.ANS_YES OR Answers.ANS_NO));
END_VAR
VAR
	Alg_Start_reset:	ph_algoritm (table:=ADR(phasesTable)):=		(phaseNumber:=0, Im:=algoritms.Test_P, act:=PhaseAlgoritmAction.run, waitCompletion:=FALSE);
END_VAR

SUPER^();
IF	NOT Alg_Start_reset.start THEN
	Start_Prov_Pusk.ask ();
END_IF
IF	(Start_Prov_Pusk.answer=Answers.ANS_YES) THEN
	algoritms.Test_P.CanRun:=TRUE;
	Alg_Start_reset.run ();
	Start_Prov_Pusk.reset ();
	reset ();
ELSIF	(Start_Prov_Pusk.answer=Answers.ANS_NO) THEN
		algoritms.Test_P.CanRun:=FALSE;
		Start_Prov_Pusk.reset ();
		reset ();
END_IF

METHOD PUBLIC reset
VAR_INPUT
END_VAR
SUPER^.reset();
Start_Prov_Pusk.reset ();
END_METHOD

END_FUNCTION_BLOCK

// K1/std12k5/Start_ALG/Start_Test_Pr
{attribute 'symbol' := 'none'}
FUNCTION_BLOCK Start_Test_Pr EXTENDS StepBySteapAlgoritm
VAR_INPUT
END_VAR
	
VAR_OUTPUT
	{attribute 'symbol' := 'read'}
	Start_Prov_Pusk:		Question(table:=ADR(ObjectTable)):=			(AnswerVariants:=(Answers.ANS_YES OR Answers.ANS_NO));
END_VAR
VAR
	Alg_Start_reset:	ph_algoritm (table:=ADR(phasesTable)):=		(phaseNumber:=0, Im:=algoritms.Test_P, act:=PhaseAlgoritmAction.run, waitCompletion:=FALSE);
END_VAR

SUPER^();
IF	NOT Alg_Start_reset.start THEN
	Start_Prov_Pusk.ask ();
END_IF
IF	(Start_Prov_Pusk.answer=Answers.ANS_YES) THEN
	algoritms.Test_P.CanRun:=TRUE;
	Alg_Start_reset.run ();
	Start_Prov_Pusk.reset ();
	reset ();
ELSIF	(Start_Prov_Pusk.answer=Answers.ANS_NO) THEN
		algoritms.Test_P.CanRun:=FALSE;
		Start_Prov_Pusk.reset ();
		reset ();
END_IF

METHOD PUBLIC reset
VAR_INPUT
END_VAR
SUPER^.reset();
Start_Prov_Pusk.reset ();
END_METHOD

END_FUNCTION_BLOCK

// K2/std12k5/Logic/AI_Final_SIP
{attribute 'symbol' := 'none'}
FUNCTION_BLOCK AI_Final_SIP EXTENDS AI_Final
VAR_INPUT
	{attribute 'symbol' := 'read'}
	ChangeSIP:AnalogParametr(table:=ADR(objectTable)):=(Value:=RNaN(), minVal:=0, maxVal:=15);
	
END_VAR
VAR_OUTPUT
END_VAR
VAR
	
END_VAR

SUPER^();
maxchangespeed:=ChangeSIP.Value;

METHOD setNewSIP
VAR_INPUT
END_VAR

maxChangeSpeed:=sip.Yst [n];


SaveToFile();
END_METHOD

END_FUNCTION_BLOCK

// K1/std12k5/Logic/AI_Final_SIP
{attribute 'symbol' := 'none'}
FUNCTION_BLOCK AI_Final_SIP EXTENDS AI_Final
VAR_INPUT
		{attribute 'symbol' := 'read'}
	ChangeSIP:AnalogParametr(table:=ADR(objectTable)):=(Value:=RNaN(), minVal:=0, maxVal:=15);
END_VAR
VAR_OUTPUT
END_VAR
VAR
	
END_VAR

SUPER^();
	maxchangespeed:=ChangeSIP.Value;

METHOD setNewSIP
VAR_INPUT
END_VAR

maxChangeSpeed:=sip.Yst [n];


SaveToFile();
END_METHOD

END_FUNCTION_BLOCK

// LowLevel_Algoritms/im/Kr4
{attribute 'symbol' := 'none'}
FUNCTION_BLOCK Kr4 EXTENDS Kran
VAR_INPUT
	
END_VAR 
VAR_OUTPUT
END_VAR
VAR
END_VAR

SUPER^();
IF im.Kr_4_Open_From_Alg.Q THEN
	sdvig:=FALSE;
END_IF

END_FUNCTION_BLOCK
